(* CODESYS project G42_assignment_2.export

Project tree, tasks and I/O mapping:
  control/
    function block door_ctrl [SFC]
    program ElevatorControl [LD]
    function block emergcy_handler [FBD]
    function block floor_request_handler [FBD]
    function block last_floor_manager [LD]
    program main [ST]
*)

// control/door_ctrl
FUNCTION_BLOCK door_ctrl
VAR_INPUT
	stopped_at_floor:BOOL;
	open_sig:BOOL;
	force_open:BOOL;
	force_close:BOOL;
	open_sensor:BOOL;
	close_sensor:BOOL;
END_VAR
VAR_OUTPUT
	open_door:BOOL;
	block_move:BOOL;
	allow_move:BOOL;
END_VAR
VAR
END_VAR

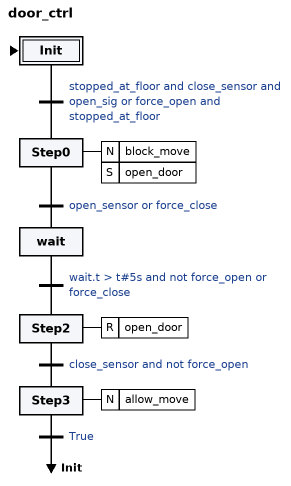
INITIAL_STEP Init:
END_STEP
TRANSITION FROM Init TO Step0
    := stopped_at_floor and close_sensor and open_sig or force_open and stopped_at_floor;
END_TRANSITION
STEP Step0:
    block_move(N);
    open_door(S);
END_STEP
TRANSITION FROM Step0 TO wait
    := open_sensor or force_close;
END_TRANSITION
STEP wait:
END_STEP
TRANSITION FROM wait TO Step2
    := wait.t > t#5s and not force_open or force_close;
END_TRANSITION
STEP Step2:
    open_door(R);
END_STEP
TRANSITION FROM Step2 TO Step3
    := close_sensor and not force_open;
END_TRANSITION
STEP Step3:
    allow_move(N);
END_STEP
TRANSITION FROM Step3 TO Init
    := True;
END_TRANSITION

END_FUNCTION_BLOCK

// control/ElevatorControl
PROGRAM ElevatorControl
VAR
	request1:BOOL;
	request2:BOOL;
	request3:BOOL;
	request4:BOOL :=TRUE;
	
	floor_request_handler:floor_request_handler;
	last_floor_manager:last_floor_manager;
	
	dorr_ctrl_1:door_ctrl;
	dorr_ctrl_2:door_ctrl;
	dorr_ctrl_3:door_ctrl;
	dorr_ctrl_4:door_ctrl;
	
	move_blocker:BOOL;
	emergency_blocker:BOOL;
	emergcy_handler:emergcy_handler;
END_VAR
VAR // added by the converter: edge detectors and wires of the graphical bodies
    _ft1, _ft2, _ft3, _ft4 : F_TRIG;
END_VAR

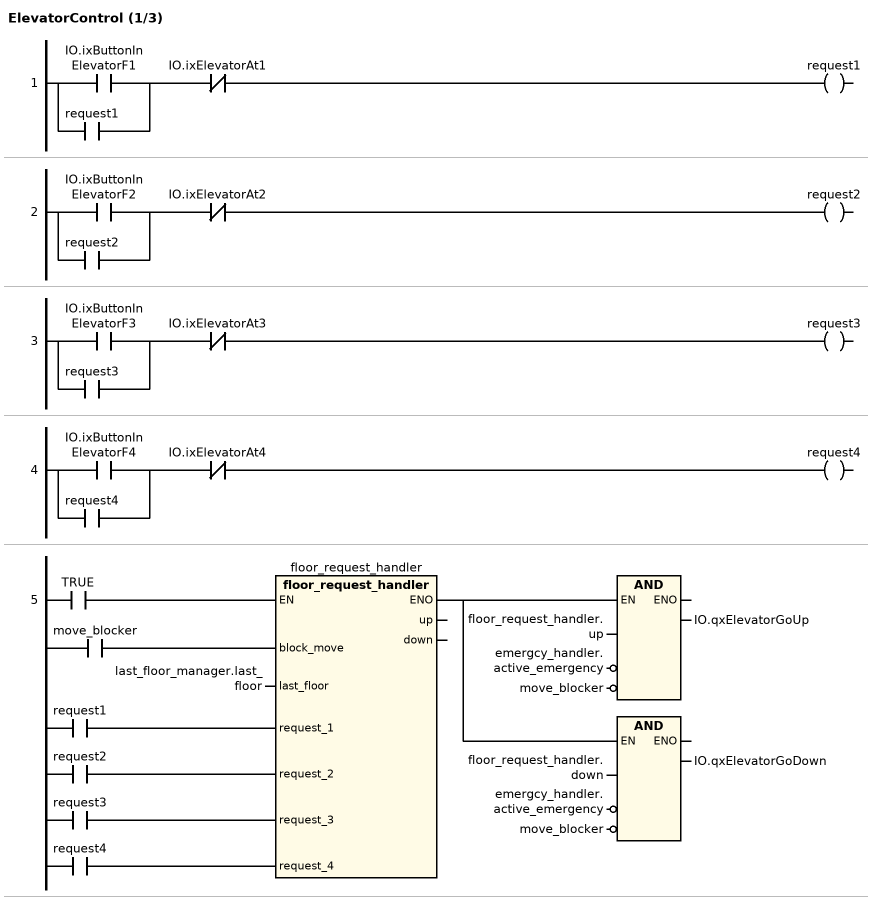
// NETWORK 1
request1 := (IO.ixButtonInElevatorF1 OR request1) AND NOT IO.ixElevatorAt1;

// NETWORK 2
request2 := (IO.ixButtonInElevatorF2 OR request2) AND NOT IO.ixElevatorAt2;

// NETWORK 3
request3 := (IO.ixButtonInElevatorF3 OR request3) AND NOT IO.ixElevatorAt3;

// NETWORK 4
request4 := (IO.ixButtonInElevatorF4 OR request4) AND NOT IO.ixElevatorAt4;

// NETWORK 5
floor_request_handler(
    block_move := move_blocker,
    last_floor := last_floor_manager.last_floor,
    request_1 := request1,
    request_2 := request2,
    request_3 := request3,
    request_4 := request4);
IO.qxElevatorGoUp := floor_request_handler.up AND NOT emergcy_handler.active_emergency AND NOT move_blocker;
IO.qxElevatorGoDown := floor_request_handler.down AND NOT emergcy_handler.active_emergency AND NOT move_blocker;

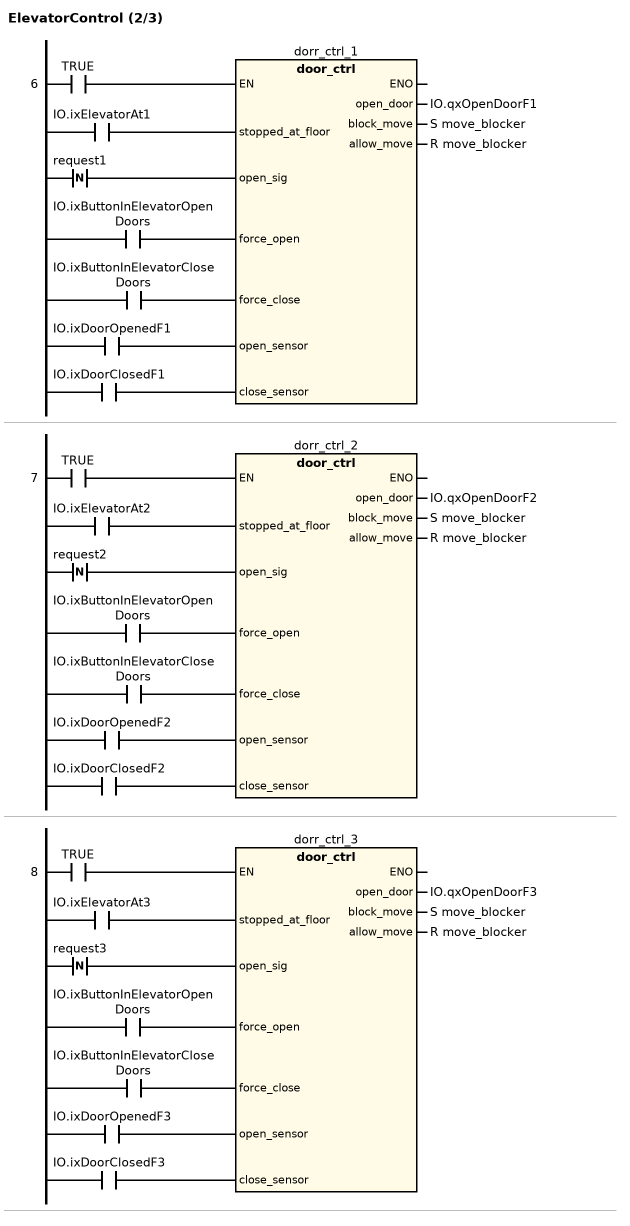
// NETWORK 6
_ft1(CLK := request1);
dorr_ctrl_1(
    stopped_at_floor := IO.ixElevatorAt1,
    open_sig := _ft1.Q,
    force_open := IO.ixButtonInElevatorOpenDoors,
    force_close := IO.ixButtonInElevatorCloseDoors,
    open_sensor := IO.ixDoorOpenedF1,
    close_sensor := IO.ixDoorClosedF1,
    open_door => IO.qxOpenDoorF1); // door_ctrl
move_blocker S= dorr_ctrl_1.block_move;
move_blocker R= dorr_ctrl_1.allow_move;

// NETWORK 7
_ft2(CLK := request2);
dorr_ctrl_2(
    stopped_at_floor := IO.ixElevatorAt2,
    open_sig := _ft2.Q,
    force_open := IO.ixButtonInElevatorOpenDoors,
    force_close := IO.ixButtonInElevatorCloseDoors,
    open_sensor := IO.ixDoorOpenedF2,
    close_sensor := IO.ixDoorClosedF2,
    open_door => IO.qxOpenDoorF2); // door_ctrl
move_blocker S= dorr_ctrl_2.block_move;
move_blocker R= dorr_ctrl_2.allow_move;

// NETWORK 8
_ft3(CLK := request3);
dorr_ctrl_3(
    stopped_at_floor := IO.ixElevatorAt3,
    open_sig := _ft3.Q,
    force_open := IO.ixButtonInElevatorOpenDoors,
    force_close := IO.ixButtonInElevatorCloseDoors,
    open_sensor := IO.ixDoorOpenedF3,
    close_sensor := IO.ixDoorClosedF3,
    open_door => IO.qxOpenDoorF3); // door_ctrl
move_blocker S= dorr_ctrl_3.block_move;
move_blocker R= dorr_ctrl_3.allow_move;

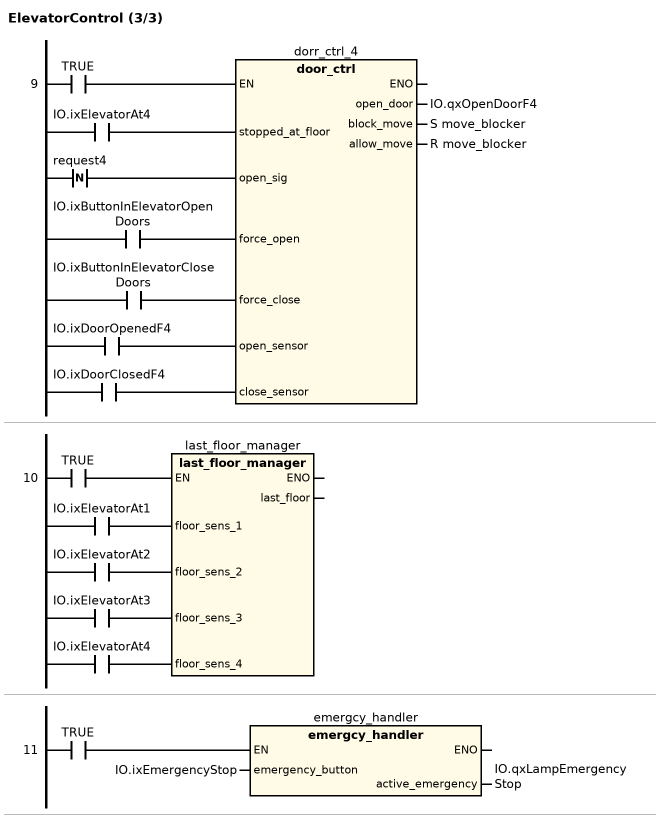
// NETWORK 9
_ft4(CLK := request4);
dorr_ctrl_4(
    stopped_at_floor := IO.ixElevatorAt4,
    open_sig := _ft4.Q,
    force_open := IO.ixButtonInElevatorOpenDoors,
    force_close := IO.ixButtonInElevatorCloseDoors,
    open_sensor := IO.ixDoorOpenedF4,
    close_sensor := IO.ixDoorClosedF4,
    open_door => IO.qxOpenDoorF4); // door_ctrl
move_blocker S= dorr_ctrl_4.block_move;
move_blocker R= dorr_ctrl_4.allow_move;

// NETWORK 10
last_floor_manager(
    floor_sens_1 := IO.ixElevatorAt1,
    floor_sens_2 := IO.ixElevatorAt2,
    floor_sens_3 := IO.ixElevatorAt3,
    floor_sens_4 := IO.ixElevatorAt4);

// NETWORK 11
emergcy_handler(emergency_button := IO.ixEmergencyStop, active_emergency => IO.qxLampEmergencyStop);

END_PROGRAM

// control/floor_request_handler
FUNCTION_BLOCK floor_request_handler
VAR_INPUT
	block_move: BOOL;
	last_floor:INT;
	request_1:BOOL;
	request_2:BOOL;
	request_3:BOOL;
	request_4:BOOL;
	
END_VAR
VAR_OUTPUT
	up:BOOL;
	down:BOOL;
END_VAR
VAR
	floor1: INT:=1;
	floor2: INT:=2;
	floor3: INT:=3;
	floor4: INT:=4;
END_VAR

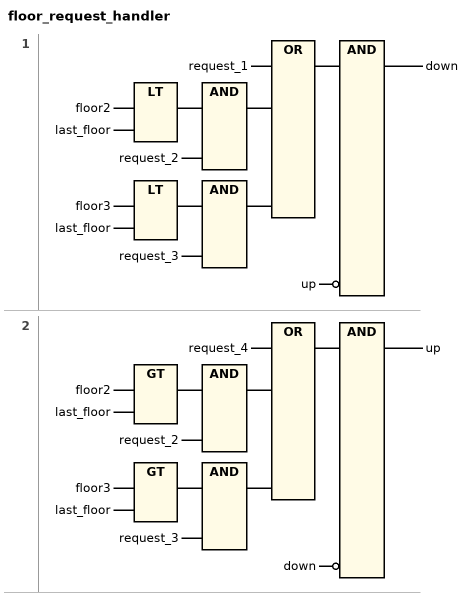
// NETWORK 1
down := (request_1 OR floor2 < last_floor AND request_2 OR floor3 < last_floor AND request_3) AND NOT up;

// NETWORK 2
up := (request_4 OR floor2 > last_floor AND request_2 OR floor3 > last_floor AND request_3) AND NOT down;

END_FUNCTION_BLOCK

// control/last_floor_manager
FUNCTION_BLOCK last_floor_manager
VAR_INPUT
	floor_sens_1:BOOL;
	floor_sens_2:BOOL;
	floor_sens_3:BOOL;
	floor_sens_4:BOOL;
END_VAR
VAR_OUTPUT
	last_floor: INT := 4;
END_VAR
VAR
END_VAR
VAR // added by the converter: edge detectors and wires of the graphical bodies
    _rt1, _rt2, _rt3, _rt4 : R_TRIG;
END_VAR

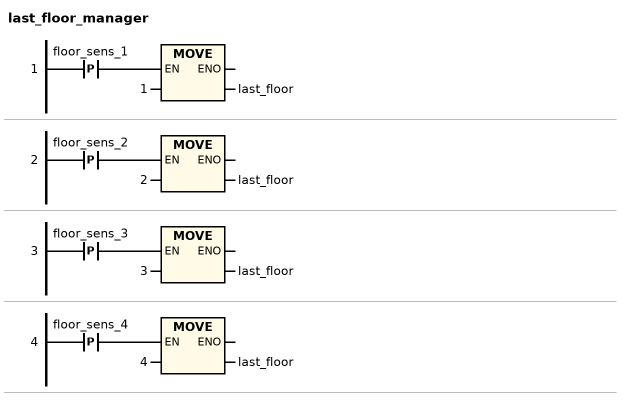
// NETWORK 1
_rt1(CLK := floor_sens_1);
IF _rt1.Q THEN last_floor := 1; END_IF

// NETWORK 2
_rt2(CLK := floor_sens_2);
IF _rt2.Q THEN last_floor := 2; END_IF

// NETWORK 3
_rt3(CLK := floor_sens_3);
IF _rt3.Q THEN last_floor := 3; END_IF

// NETWORK 4
_rt4(CLK := floor_sens_4);
IF _rt4.Q THEN last_floor := 4; END_IF

END_FUNCTION_BLOCK

// control/emergcy_handler
FUNCTION_BLOCK emergcy_handler
VAR_INPUT
	emergency_button:BOOL;
END_VAR
VAR_OUTPUT
	active_emergency: BOOL;
END_VAR
VAR
	timer : TON;
	
END_VAR
VAR // added by the converter: edge detectors and wires of the graphical bodies
    _rt1 : R_TRIG;
END_VAR

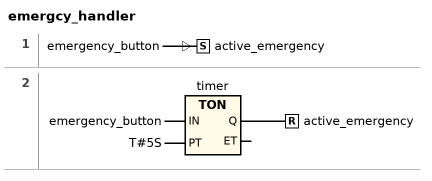
// NETWORK 1
_rt1(CLK := emergency_button);
active_emergency S= _rt1.Q;

// NETWORK 2
timer(IN := emergency_button, PT := T#5S); // TON
active_emergency R= timer.Q;

END_FUNCTION_BLOCK

// control/main
PROGRAM main
VAR
END_VAR

ElevatorControl();

END_PROGRAM
